// This function has been automatically generated from the project information.
{attribute 'signature_flag' := '1073741824'}
{attribute 'TcGenerated'}
{attribute 'no-analysis'}
FUNCTION F_GetCompany : WSTRING
VAR_INPUT
	
END_VAR

F_GetCompany := "Daniel Wiege";

END_FUNCTION

(* stored: Version 1.1.0.1
   POU F_GetCompany: Id {4f584e42-e9f1-43cf-ac45-443db7cd1273}, SpecialFunc None *)
